// TwinCAT 3 PLC project Baustromverteiler
// ProgramVersion: 3.1.4023.0
// libraries:
//   EfficientIO Communicator, * (EfficientIO)
//   Lynus Energy Basic, * (Lynus AG)
//   Lynus Standards, * (Lynus AG)
//   Tc2_BABasic, * (Beckhoff Automation GmbH)
//   Tc2_Standard, * (Beckhoff Automation GmbH)
//   Tc2_System, * (Beckhoff Automation GmbH)
//   Tc2_Utilities, * (Beckhoff Automation GmbH)
//   Tc3_IotBase, * (Beckhoff Automation GmbH)
//   Tc3_JsonXml, * (Beckhoff Automation GmbH)
//   Tc3_Module, * (Beckhoff Automation GmbH)
// project tree:
//   / FastTask.TcTTO (not stored), GlobalTextList.TcGTLO, MiddleTask.TcTTO, SlowTask.TcTTO (not stored)
//   FBs/ FB_Enphase.TcPOU, FB_Enphase_Helper.TcPOU, FB_Shelly_Pro4PM.TcPOU, FB_Shelly_Pro4PM_Helper.TcPOU
//   POUs/ prgContactors.TcPOU, prgEM.TcPOU, prgEnphase.TcPOU, prgGrid.TcPOU, prgShelly1.TcPOU, prgShelly2.TcPOU, prgComEffIO.TcPOU, prgRWEffIO.TcPOU, prgSystemTime.TcPOU, prgVarEffIO.TcPOU (not stored)
// real-time tasks:
//   TASK FastTask: cycle T#5ms, priority 6, ADS port 350
//   TASK MiddleTask: cycle T#10ms, priority 8, ADS port 351
//   TASK SlowTask: cycle T#20ms, priority 10, ADS port 352
// I/O:
//   DEVICE Device 1 (Beckhoff CCAT)
//   DEVICE Device 2 (CX-BK)
//     Box 1 (CX-BK)
// variable links:
//   Baustromverteiler/Baustromverteiler Instance <-> Device 2 (CX-BK)/Box 1 (CX-BK)
//     MiddleTask Inputs/prgEM.fbEM1.fbKL3403.byStateCH1 <-> Term 3 (KL3403)/Channel 1/State
//     MiddleTask Inputs/prgEM.fbEM1.fbKL3403.byStateCH2 <-> Term 3 (KL3403)/Channel 2/State
//     MiddleTask Inputs/prgEM.fbEM1.fbKL3403.byStateCH3 <-> Term 3 (KL3403)/Channel 3/State
//     MiddleTask Inputs/prgEM.fbEM3.fbKL3403.byStateCH1 <-> Term 5 (KL3403)/Channel 1/State
//     MiddleTask Inputs/prgEM.fbEM3.fbKL3403.byStateCH2 <-> Term 5 (KL3403)/Channel 2/State
//     MiddleTask Inputs/prgEM.fbEM3.fbKL3403.byStateCH3 <-> Term 5 (KL3403)/Channel 3/State
//     MiddleTask Inputs/prgEM.fbEM1.fbKL3403.iDataInCH1 <-> Term 3 (KL3403)/Channel 1/Data In
//     MiddleTask Inputs/prgEM.fbEM1.fbKL3403.iDataInCH2 <-> Term 3 (KL3403)/Channel 2/Data In
//     MiddleTask Inputs/prgEM.fbEM1.fbKL3403.iDataInCH3 <-> Term 3 (KL3403)/Channel 3/Data In
//     MiddleTask Inputs/prgEM.fbEM3.fbKL3403.iDataInCH1 <-> Term 5 (KL3403)/Channel 1/Data In
//     MiddleTask Inputs/prgEM.fbEM3.fbKL3403.iDataInCH2 <-> Term 5 (KL3403)/Channel 2/Data In
//     MiddleTask Inputs/prgEM.fbEM3.fbKL3403.iDataInCH3 <-> Term 5 (KL3403)/Channel 3/Data In
//     MiddleTask Inputs/prgEM.fbKBusState.uiKBusState_OUT <-> Inputs/State
//     MiddleTask Outputs/prgContactors.bCircle6Switch <-> Term 2 (KL2408)/Channel 1/Output
//     MiddleTask Outputs/prgContactors.bCircle7Switch <-> Term 2 (KL2408)/Channel 3/Output
//     MiddleTask Outputs/prgEM.fbEM1.fbKL3403.byCntrCH1 <-> Term 3 (KL3403)/Channel 1/Ctrl
//     MiddleTask Outputs/prgEM.fbEM1.fbKL3403.byCntrCH2 <-> Term 3 (KL3403)/Channel 2/Ctrl
//     MiddleTask Outputs/prgEM.fbEM1.fbKL3403.byCntrCH3 <-> Term 3 (KL3403)/Channel 3/Ctrl
//     MiddleTask Outputs/prgEM.fbEM3.fbKL3403.byCntrCH1 <-> Term 5 (KL3403)/Channel 1/Ctrl
//     MiddleTask Outputs/prgEM.fbEM3.fbKL3403.byCntrCH2 <-> Term 5 (KL3403)/Channel 2/Ctrl
//     MiddleTask Outputs/prgEM.fbEM3.fbKL3403.byCntrCH3 <-> Term 5 (KL3403)/Channel 3/Ctrl

CONFIGURATION Baustromverteiler
    RESOURCE PLC ON TwinCAT3
        TASK MiddleTask(INTERVAL := T#10ms, PRIORITY := 8);
        PROGRAM prgContactors WITH MiddleTask : prgContactors;
        PROGRAM prgEM WITH MiddleTask : prgEM;
        PROGRAM prgShelly1 WITH MiddleTask : prgShelly1;
        PROGRAM prgShelly2 WITH MiddleTask : prgShelly2;
        PROGRAM prgSystemTime WITH MiddleTask : prgSystemTime;
        PROGRAM prgEnphase WITH MiddleTask : prgEnphase;
        PROGRAM prgGrid WITH MiddleTask : prgGrid;
    END_RESOURCE
END_CONFIGURATION

// ---- POUs/prgContactors.TcPOU
PROGRAM prgContactors
VAR
	bCircle6On				: BOOL;						//{#lynus.ag#()}
	bCircle6Off				: BOOL;						//{#lynus.ag#()}
	bCircle7On				: BOOL;						//{#lynus.ag#()}
	bCircle7Off				: BOOL;						//{#lynus.ag#()}
	bCircle6Switch	AT%Q*	: BOOL;						//{#lynus.ag#()}
	bCircle7Switch	AT%Q*	: BOOL;						//{#lynus.ag#()}
	fbCircle6				: FB_Light;
	fbCircle7				: FB_Light;
END_VAR

fbCircle6(bOn:=bCircle6On, bOff:=bCircle6Off, bLight=>bCircle6Switch);

fbCircle7(bOn:=bCircle7On, bOff:=bCircle7Off, bLight=>bCircle7Switch);

END_PROGRAM

// ---- POUs/prgEM.TcPOU
PROGRAM prgEM
VAR
	fbKBusState		: FB_K_Bus_State;
	fbEM1			: FB_EM_Beckhoff_KL3403;
	fbEM1Counter	: FB_EnergyCounter;
	fbEM2			: FB_EM_Beckhoff_KL3403;
	fbEM2Counter	: FB_EnergyCounter;
	fbEM3			: FB_EM_Beckhoff_KL3403;
	fbEM3Counter	: FB_EnergyCounter;
	fbC5Counter		: FB_EnergyCounter;
	lrPowerEM1		: LREAL;						//{#lynus.ag#()}
	lrPowerEM2		: LREAL;						//{#lynus.ag#()}
	lrPowerEM3		: LREAL;						//{#lynus.ag#()}
	lrPowerC5		: LREAL;						//{#lynus.ag#()}
END_VAR
VAR PERSISTENT
	lrCounterEM1	: LREAL;						//{#lynus.ag#()}
	lrCounterEM2	: LREAL;						//{#lynus.ag#()}
	lrCounterEM3	: LREAL;						//{#lynus.ag#()}
	lrCounterC5		: LREAL;						//{#lynus.ag#()}
END_VAR

fbKBusState(uiKBusState_OUT=> );

// Base Connection

fbEM1(
	bEnable:= TRUE, 
	bChannel1Invers:= TRUE,
	bChannel2Invers:= TRUE,
	bChannel3Invers:= TRUE,
	uiCurrentTransformerRatioL1:= 64, 
	uiCurrentTransformerRatioL2:= 64, 
	uiCurrentTransformerRatioL3:= 64, 
	uiKBusState_IN:= fbKBusState.uiKBusState_OUT, 
	stDataEMPower=> , 
	stDataEMCounter=> , 
	stDataEMPowerRealTime=> , 
	stDataEMCounterRealTime=> , 
	diNrOfEM_OUT=> );

lrPowerEM1 := fbEM1.stDataEMPower.lrPowerTotal;	

fbEM1Counter(
	byActiveTariff:= 1, 
	lrPowerInput:= lrPowerEM1, 
	lrTotalCounterEnergy_Consumption=> , 
	lrTotalCounterEnergy_Production=> , 
	lrCounterEnergyT1_Consumption=> , 
	lrCounterEnergyT2_Consumption=> , 
	lrCounterEnergyT1_Production=> , 
	lrCounterEnergyT2_Production=> );
	
IF fbEM1Counter.lrTotalCounterEnergy_Consumption > lrCounterEM1 THEN  	
	lrCounterEM1 := fbEM1Counter.lrTotalCounterEnergy_Consumption;
END_IF


// Circle6, 400V/32A

fbEM2(
	bEnable:= TRUE, 
	bChannel1Invers:= TRUE,
	bChannel2Invers:= TRUE,
	bChannel3Invers:= TRUE,
	uiCurrentTransformerRatioL1:= 35, 
	uiCurrentTransformerRatioL2:= 35, 
	uiCurrentTransformerRatioL3:= 35, 
	uiKBusState_IN:= fbKBusState.uiKBusState_OUT, 
	stDataEMPower=> , 
	stDataEMCounter=> , 
	stDataEMPowerRealTime=> , 
	stDataEMCounterRealTime=> , 
	diNrOfEM_OUT=> );

lrPowerEM2 := fbEM2.stDataEMPower.lrPowerTotal;	

fbEM2Counter(
	byActiveTariff:= 1, 
	lrPowerInput:= lrPowerEM2, 
	lrTotalCounterEnergy_Consumption=> , 
	lrTotalCounterEnergy_Production=> , 
	lrCounterEnergyT1_Consumption=> , 
	lrCounterEnergyT2_Consumption=> , 
	lrCounterEnergyT1_Production=> , 
	lrCounterEnergyT2_Production=> );
	
IF fbEM2Counter.lrTotalCounterEnergy_Consumption > lrCounterEM2 THEN  	
	lrCounterEM2 := fbEM2Counter.lrTotalCounterEnergy_Consumption;
END_IF


// Circle7, 400V/32A

fbEM3(
	bEnable:= TRUE, 
	bChannel1Invers:= FALSE,
	bChannel2Invers:= FALSE,
	bChannel3Invers:= FALSE,
	uiCurrentTransformerRatioL1:= 100, 
	uiCurrentTransformerRatioL2:= 100, 
	uiCurrentTransformerRatioL3:= 100, 
	uiKBusState_IN:= fbKBusState.uiKBusState_OUT, 
	stDataEMPower=> , 
	stDataEMCounter=> , 
	stDataEMPowerRealTime=> , 
	stDataEMCounterRealTime=> , 
	diNrOfEM_OUT=> );

lrPowerEM3 := fbEM3.stDataEMPower.lrPowerTotal;	

fbEM3Counter(
	byActiveTariff:= 1, 
	lrPowerInput:= lrPowerEM3, 
	lrTotalCounterEnergy_Consumption=> , 
	lrTotalCounterEnergy_Production=> , 
	lrCounterEnergyT1_Consumption=> , 
	lrCounterEnergyT2_Consumption=> , 
	lrCounterEnergyT1_Production=> , 
	lrCounterEnergyT2_Production=> );
	
IF fbEM3Counter.lrTotalCounterEnergy_Consumption > lrCounterEM3 THEN  	
	lrCounterEM3 := fbEM3Counter.lrTotalCounterEnergy_Consumption;
END_IF


// Circle5, 400V/16A

IF lrPowerEM1 - (lrPowerEM2 + lrPowerEM3 + prgShelly1.lrPowerC1 + prgShelly1.lrPowerC2 + prgShelly2.lrPowerC3 + prgShelly2.lrPowerC4) >= 0 THEN  	
	lrPowerC5 := lrPowerEM1 - (lrPowerEM2 + lrPowerEM3 + prgShelly1.lrPowerC1 + prgShelly1.lrPowerC2 + prgShelly2.lrPowerC3 + prgShelly2.lrPowerC4);
	ELSE
		lrPowerC5 := 0;
END_IF

fbC5Counter(
	byActiveTariff:= 1, 
	lrPowerInput:= lrPowerC5, 
	lrTotalCounterEnergy_Consumption=> , 
	lrTotalCounterEnergy_Production=> , 
	lrCounterEnergyT1_Consumption=> , 
	lrCounterEnergyT2_Consumption=> , 
	lrCounterEnergyT1_Production=> , 
	lrCounterEnergyT2_Production=> );
	
IF fbC5Counter.lrTotalCounterEnergy_Consumption > lrCounterC5 THEN  	
	lrCounterC5 := fbC5Counter.lrTotalCounterEnergy_Consumption;
END_IF

END_PROGRAM

// ---- POUs/prgShelly1.TcPOU
PROGRAM prgShelly1
VAR
	fbShelly1					: FB_Shelly_Pro4PM;
	// Circle1, 230V
	lrPowerC1					: LREAL;	//{#lynus.ag#()}
	lrVoltageC1					: LREAL;	//{#lynus.ag#()}
	lrEnergyC1					: LREAL;	//{#lynus.ag#()}
	lrPowerC1_W					: LREAL;
	lrEnergyC1_Wh				: LREAL;
	bCircle1On					: BOOL;		//{#lynus.ag#()}
	bCircle1Off					: BOOL;		//{#lynus.ag#()}
	bCircle1Switch				: BOOL;		//{#lynus.ag#()}

	// Circle2, 230V
	lrPowerC2					: LREAL;	//{#lynus.ag#()}
	lrVoltageC2					: LREAL;	//{#lynus.ag#()}
	lrEnergyC2					: LREAL;	//{#lynus.ag#()}
	lrPowerC2_W					: LREAL;
	lrEnergyC2_Wh				: LREAL;
	bCircle2On					: BOOL;		//{#lynus.ag#()}
	bCircle2Off					: BOOL;		//{#lynus.ag#()}
	bCircle2Switch				: BOOL;		//{#lynus.ag#()}
END_VAR

VAR PERSISTENT
// trigger command execution
	bEnableShelly1				: BOOL;		//{#lynus.ag#()}
END_VAR

fbShelly1(
	bStart:= bEnableShelly1, 
	tDelayRequest:= T#3S, 
	sHostname:= '192.168.1.20', 
	bValidResult=> , 
	bBusy=> , 
	bError=> , 
	bDone=> , 
	hrErrorCode=> ,
	lrpowerP1=> lrPowerC1_W, 
	lrvoltageP1=> lrVoltageC1, 
	lrenergyP1=> lrEnergyC1_Wh,
	lrpowerP2=> lrPowerC2_W, 
	lrvoltageP2=> lrVoltageC2, 
	lrenergyP2=> lrEnergyC2_Wh,
	bOnP1:= bCircle1On,
	bOffP1:= bCircle1Off,
	bStateP1=> bCircle1Switch,
	bOnP2:= bCircle2On,
	bOffP2:= bCircle2Off,
	bStateP2=> bCircle2Switch );

// re-calc Power to kW / kWh
lrPowerC1 := lrPowerC1_W / 1000;
lrPowerC2 := lrPowerC2_W / 1000;
lrEnergyC1 := lrEnergyC1_Wh / 1000;
lrEnergyC2 := lrEnergyC2_Wh / 1000;

END_PROGRAM

// ---- FBs/FB_Shelly_Pro4PM.TcPOU
FUNCTION_BLOCK FB_Shelly_Pro4PM
VAR_INPUT
	bStart				: BOOL;
	tDelayRequest		: TIME := T#3S;		//Timer for delay before start with the next read or write Request
	sHostname			: STRING(255);		//Hostname or IP Adress from the Server
	bOnP1				: BOOL;
	bOffP1				: BOOL;
	bOnP2				: BOOL;
	bOffP2				: BOOL;
	bOnP3				: BOOL;
	bOffP3				: BOOL;
	bOnP4				: BOOL;
	bOffP4				: BOOL;
END_VAR

VAR_IN_OUT
END_VAR

VAR_OUTPUT
	bValidResult				: BOOL;															//Valid Result received from Server
    bBusy						: BOOL;															//Function is Busy
    bError						: BOOL;															//Error sucess
	bDone						: BOOL;															//True after the decoding from the received Json File
	bConnected					: BOOL;															//Connection to the Server
	lrpowerP1					: LREAL;														//Received Value
	lrvoltageP1					: LREAL;														//Received Value
	lrenergyP1					: LREAL;														//Received Value
	lrpowerP2					: LREAL;														//Received Value
	lrvoltageP2					: LREAL;														//Received Value
	lrenergyP2					: LREAL;
	lrpowerP3					: LREAL;														//Received Value
	lrvoltageP3					: LREAL;														//Received Value
	lrenergyP3					: LREAL;
	lrpowerP4					: LREAL;														//Received Value
	lrvoltageP4					: LREAL;														//Received Value
	lrenergyP4					: LREAL;	
	hrErrorCode       			: HRESULT;														//Error Result from Http Client
	bStateP1					: BOOL;
	bStateP2					: BOOL;
	bStateP3					: BOOL;
	bStateP4					: BOOL;
END_VAR

VAR
	fbClient					: FB_IotHttpClient;
	fbHttpGet					: FB_Shelly_Pro4PM_Helper;
	timStartRequest				: TON;															//Timer to Start the Request
	FPStartRequest				: R_TRIG;														//Internal positive Edge
	FPDone						: R_TRIG;														//Internal positive Edge
	FNStart						: F_TRIG;														//Internal negative Edge
	SwitchOnP1					: R_TRIG;
	SwitchOffP1					: R_TRIG;
	SwitchOnP2					: R_TRIG;
	SwitchOffP2					: R_TRIG;
	SwitchOnP3					: R_TRIG;
	SwitchOffP3					: R_TRIG;
	SwitchOnP4					: R_TRIG;
	SwitchOffP4					: R_TRIG;
END_VAR

(*------------------------------------------------------------------------------------Configure HTTP Client------------------------------------------------------------------------------------------------------*)

fbClient.sHostName := sHostname;
fbClient.tConnectionTimeout := tDelayRequest;

IF NOT fbClient.bConfigured THEN 
	fbClient.nHostPort:= 80;
	fbClient.bKeepAlive := TRUE;
	fbClient.tConnectionTimeout := T#2S;
END_IF


//Timer to start the Request
FPStartRequest(CLK:= bStart, Q=> );
	timStartRequest(IN:= fbClient.bConfigured AND bStart AND NOT timStartRequest.Q, PT:= tDelayRequest, Q=> , ET=> );
		IF ((timStartRequest.Q AND NOT bBusy) OR (FPStartRequest.Q AND NOT bBusy AND fbClient.bConfigured)) THEN fbHttpGet.bSend := TRUE; END_IF

				
//Http Get Function
fbHttpGet(
	lrapowerP1 => lrpowerP1, 
	lrvoltageP1 => lrvoltageP1, 
	lraenergyP1 => lrenergyP1,
	lrapowerP2 => lrpowerP2, 
	lrvoltageP2 => lrvoltageP2, 
	lraenergyP2 => lrenergyP2,
	lrapowerP3 => lrpowerP3, 
	lrvoltageP3 => lrvoltageP3, 
	lraenergyP3 => lrenergyP3,
	lrapowerP4 => lrpowerP4, 
	lrvoltageP4 => lrvoltageP4, 
	lraenergyP4 => lrenergyP4, 
	bSend:= , 
	fbClient:= fbClient, 
	bBusy=> bBusy, 
	bError=> ,
	sContentS0=> ,
	sContentS1=> ,
	sContentS2=> ,
	sContentS3=> ,
	bStateP1=>bStateP1,
	bStateP2=>bStateP2,
	bStateP3=>bStateP3,
	bStateP4=>bStateP4 );


fbHttpGet.bSend := FALSE;

FPDone(CLK:= bDone, Q=> );

(*
//Http Client
FNStart(CLK:= bStart, Q=> );
	IF FNStart.Q THEN fbClient.Disconnect(); END_IF
*)

fbClient.Execute();

//Error
IF fbHttpGet.bError OR fbClient.bError THEN bError := TRUE; ELSE bError := FALSE; END_IF	
	hrErrorCode := fbClient.hrErrorCode;
	

// Relay Control, Switch P1
SwitchOnP1(CLK:=bOnP1);
IF SwitchOnP1.Q THEN
	fbHttpGet.bSetOnP1 := TRUE;
END_IF

SwitchOffP1(CLK:=bOffP1);
IF SwitchOffP1.Q THEN
	fbHttpGet.bSetOffP1 := TRUE;
END_IF

// Relay Control, Switch P2
SwitchOnP2(CLK:=bOnP2);
IF SwitchOnP2.Q THEN
	fbHttpGet.bSetOnP2 := TRUE;
END_IF

SwitchOffP2(CLK:=bOffP2);
IF SwitchOffP2.Q THEN
	fbHttpGet.bSetOffP2 := TRUE;
END_IF

// Relay Control, Switch P3
SwitchOnP3(CLK:=bOnP3);
IF SwitchOnP3.Q THEN
	fbHttpGet.bSetOnP3 := TRUE;
END_IF

SwitchOffP3(CLK:=bOffP3);
IF SwitchOffP3.Q THEN
	fbHttpGet.bSetOffP3 := TRUE;
END_IF

// Relay Control, Switch P4
SwitchOnP4(CLK:=bOnP4);
IF SwitchOnP4.Q THEN
	fbHttpGet.bSetOnP4 := TRUE;
END_IF

SwitchOffP4(CLK:=bOffP4);
IF SwitchOffP4.Q THEN
	fbHttpGet.bSetOffP4 := TRUE;
END_IF

END_FUNCTION_BLOCK

// ---- FBs/FB_Shelly_Pro4PM_Helper.TcPOU
FUNCTION_BLOCK FB_Shelly_Pro4PM_Helper
VAR_INPUT
	bSend			: BOOL;
	bSetOnP1		: BOOL;
	bSetOffP1		: BOOL;
	bSetOnP2		: BOOL;
	bSetOffP2		: BOOL;
	bSetOnP3		: BOOL;
	bSetOffP3		: BOOL;
	bSetOnP4		: BOOL;
	bSetOffP4		: BOOL;
END_VAR

VAR_IN_OUT
	fbClient		: FB_IotHttpClient;
END_VAR

VAR_OUTPUT
	bBusy			: BOOL;
	bError			: BOOL;
	bStateP1		: BOOL;
	bStateP2		: BOOL;
	bStateP3		: BOOL;
	bStateP4		: BOOL;
	lrapowerP1		: LREAL;
	lrvoltageP1		: LREAL;
	lraenergyP1		: LREAL;
	lrapowerP2		: LREAL;
	lrvoltageP2		: LREAL;
	lraenergyP2		: LREAL;
	lrapowerP3		: LREAL;
	lrvoltageP3		: LREAL;
	lraenergyP3		: LREAL;
	lrapowerP4		: LREAL;
	lrvoltageP4		: LREAL;
	lraenergyP4		: LREAL;
END_VAR

VAR
	fbRequestSwitch0	: FB_IotHttpRequest;
	fbRequestSwitch1	: FB_IotHttpRequest;
	fbRequestSwitch2	: FB_IotHttpRequest;
	fbRequestSwitch3	: FB_IotHttpRequest;
	fbJson				: FB_JsonDomParser;
	nState				: UDINT;
	RisingEdge			: R_TRIG;
	RisingEdgeSetOnP1	: R_TRIG;
	RisingEdgeSetOffP1	: R_TRIG;
	RisingEdgeSetOnP2	: R_TRIG;
	RisingEdgeSetOffP2	: R_TRIG;
	RisingEdgeSetOnP3	: R_TRIG;
	RisingEdgeSetOffP3	: R_TRIG;
	RisingEdgeSetOnP4	: R_TRIG;
	RisingEdgeSetOffP4	: R_TRIG;
	timTimeout			: TON;
	tTimeOut			: TIME := T#30S;
	timTimeoutSwitch	: TON;
	tTimeOutSwitch		: TIME := T#5S;
	
	bGetContentResult	: BOOL;
	sContentS0			: STRING(511);
	sContentS1			: STRING(511);
	sContentS2			: STRING(511);
	sContentS3			: STRING(511);
	
	bGetJsonResult		: BOOL;
	jsonDoc				: SJsonValue;
	jsonVal				: SJsonValue;
	
	nReqCount			: UDINT;	
	nResCount			: UDINT;
	nValidResCount		: UDINT;
	nErrCount			: UDINT;
END_VAR

//Timer for Timeout
timTimeout(IN:= nState = 1 AND bBusy, PT:= tTimeOut, Q=> , ET=> );
	IF timTimeout.Q THEN 
		nState := 0;
		bBusy := FALSE;
	END_IF
	
timTimeoutSwitch(IN:= bSetOnP1 OR bSetOffP1 OR bSetOnP2 OR bSetOffP2 OR bSetOnP3 OR bSetOffP3 OR bSetOnP4 OR bSetOffP4, PT:= tTimeOut, Q=> , ET=> );
	IF timTimeoutSwitch.Q THEN 
		bSetOnP1 := FALSE;
		bSetOffP1 := FALSE;
		bSetOnP2 := FALSE;
		bSetOffP2 := FALSE;
		bSetOnP3 := FALSE;
		bSetOffP3 := FALSE;
		bSetOnP4 := FALSE;
		bSetOffP4 := FALSE;
	END_IF

RisingEdge(CLK:= bSend );
RisingEdgeSetOnP1(CLK:= bSetOnP1 );
RisingEdgeSetOffP1(CLK:= bSetOffP1 );
RisingEdgeSetOnP2(CLK:= bSetOnP2 );
RisingEdgeSetOffP2(CLK:= bSetOffP2 );
RisingEdgeSetOnP3(CLK:= bSetOnP3 );
RisingEdgeSetOffP3(CLK:= bSetOffP3 );
RisingEdgeSetOnP4(CLK:= bSetOnP4 );
RisingEdgeSetOffP4(CLK:= bSetOffP4 );

CASE nState OF
0:	
	IF RisingEdge.Q THEN 
		IF
			fbRequestSwitch0.SendRequest(sUri:='/rpc/Switch.GetStatus?id=0', fbClient:=fbClient, eRequestType:=ETcIotHttpRequestType.HTTP_Get, 0, 0, 0) AND
			fbRequestSwitch1.SendRequest(sUri:='/rpc/Switch.GetStatus?id=1', fbClient:=fbClient, eRequestType:=ETcIotHttpRequestType.HTTP_Get, 0, 0, 0) AND
			fbRequestSwitch2.SendRequest(sUri:='/rpc/Switch.GetStatus?id=2', fbClient:=fbClient, eRequestType:=ETcIotHttpRequestType.HTTP_Get, 0, 0, 0) AND
			fbRequestSwitch3.SendRequest(sUri:='/rpc/Switch.GetStatus?id=3', fbClient:=fbClient, eRequestType:=ETcIotHttpRequestType.HTTP_Get, 0, 0, 0) THEN				
			nState:= 1;
			nReqCount:= nReqCount+1;
			bBusy:= TRUE;
			bError:= FALSE;
		END_IF					
	END_IF
	
	IF RisingEdgeSetOnP1.Q THEN 
		IF
			fbRequestSwitch0.SendRequest(sUri:='/rpc/Switch.Set?id=0&on=true', fbClient:=fbClient, eRequestType:=ETcIotHttpRequestType.HTTP_Get, 0, 0, 0) THEN				
			bSetOnP1 := FALSE;
			nState:= 1;
			bBusy:= TRUE;
			bError:= FALSE;
		END_IF					
	END_IF
	
	IF RisingEdgeSetOffP1.Q THEN 
		IF
			fbRequestSwitch0.SendRequest(sUri:='/rpc/Switch.Set?id=0&on=false', fbClient:=fbClient, eRequestType:=ETcIotHttpRequestType.HTTP_Get, 0, 0, 0) THEN				
			bSetOffP1 := FALSE;
			nState:= 1;
			bBusy:= TRUE;
			bError:= FALSE;
		END_IF					
	END_IF
	
	IF RisingEdgeSetOnP2.Q THEN 
		IF
			fbRequestSwitch1.SendRequest(sUri:='/rpc/Switch.Set?id=1&on=true', fbClient:=fbClient, eRequestType:=ETcIotHttpRequestType.HTTP_Get, 0, 0, 0) THEN				
			bSetOnP2 := FALSE;
			nState:= 1;
			bBusy:= TRUE;
			bError:= FALSE;
		END_IF					
	END_IF
	
	IF RisingEdgeSetOffP2.Q THEN 
		IF
			fbRequestSwitch1.SendRequest(sUri:='/rpc/Switch.Set?id=1&on=false', fbClient:=fbClient, eRequestType:=ETcIotHttpRequestType.HTTP_Get, 0, 0, 0) THEN				
			bSetOffP2 := FALSE;
			nState:= 1;
			bBusy:= TRUE;
			bError:= FALSE;
		END_IF					
	END_IF
	
	IF RisingEdgeSetOnP3.Q THEN 
		IF
			fbRequestSwitch2.SendRequest(sUri:='/rpc/Switch.Set?id=2&on=true', fbClient:=fbClient, eRequestType:=ETcIotHttpRequestType.HTTP_Get, 0, 0, 0) THEN				
			bSetOnP3 := FALSE;
			nState:= 1;
			bBusy:= TRUE;
			bError:= FALSE;
		END_IF					
	END_IF
	
	IF RisingEdgeSetOffP3.Q THEN 
		IF
			fbRequestSwitch2.SendRequest(sUri:='/rpc/Switch.Set?id=2&on=false', fbClient:=fbClient, eRequestType:=ETcIotHttpRequestType.HTTP_Get, 0, 0, 0) THEN				
			bSetOffP3 := FALSE;
			nState:= 1;
			bBusy:= TRUE;
			bError:= FALSE;
		END_IF					
	END_IF
	
	IF RisingEdgeSetOnP4.Q THEN 
		IF
			fbRequestSwitch3.SendRequest(sUri:='/rpc/Switch.Set?id=3&on=true', fbClient:=fbClient, eRequestType:=ETcIotHttpRequestType.HTTP_Get, 0, 0, 0) THEN				
			bSetOnP4 := FALSE;
			nState:= 1;
			bBusy:= TRUE;
			bError:= FALSE;
		END_IF					
	END_IF
	
	IF RisingEdgeSetOffP4.Q THEN 
		IF
			fbRequestSwitch3.SendRequest(sUri:='/rpc/Switch.Set?id=3&on=false', fbClient:=fbClient, eRequestType:=ETcIotHttpRequestType.HTTP_Get, 0, 0, 0) THEN				
			bSetOffP4 := FALSE;
			nState:= 1;
			bBusy:= TRUE;
			bError:= FALSE;
		END_IF					
	END_IF
	
1:
	IF NOT fbRequestSwitch0.bBusy AND NOT fbRequestSwitch1.bBusy AND NOT fbRequestSwitch2.bBusy AND NOT fbRequestSwitch3.bBusy THEN
		bError:= TRUE;
		
		IF NOT fbRequestSwitch0.bError THEN				 
			bGetContentResult:= fbRequestSwitch0.GetContent(pContent:= ADR(sContentS0), nContentSize:= SIZEOF(sContentS0), bSetNullTermination:= TRUE);
			IF fbRequestSwitch0.nStatusCode >= 200 AND fbRequestSwitch0.nStatusCode < 300 THEN
				bGetJsonResult:= FALSE;
				jsonDoc:= fbRequestSwitch0.GetJsonDomContent(fbJson);
				IF jsonDoc <> 0 THEN
					bGetJsonResult:= TRUE;
					IF fbJson.HasMember(jsonDoc, 'output')  THEN
						jsonVal:= fbJson.FindMember(jsonDoc, 'output');
						nValidResCount:= nValidResCount+1;					
						IF fbJson.IsBool(jsonVal) THEN							
							bStateP1:= fbJson.GetBool(jsonVal);									
						END_IF
						jsonVal:= fbJson.FindMember(jsonDoc, 'apower');
						nValidResCount:= nValidResCount+1;
						IF fbJson.IsDouble(jsonVal) THEN							
							lrapowerP1:= fbJson.GetDouble(jsonVal);									
						END_IF
						jsonVal:= fbJson.FindMember(jsonDoc, 'voltage');
						nValidResCount:= nValidResCount+1;					
						IF fbJson.IsDouble(jsonVal) THEN							
							lrvoltageP1:= fbJson.GetDouble(jsonVal);									
						END_IF
						jsonVal:= fbJson.FindMember(jsonDoc, 'aenergy');
                        IF fbJson.HasMember(jsonVal, 'total') THEN
                            jsonVal:= fbJson.FindMember(jsonVal, 'total');
                            nValidResCount:= nValidResCount+1;
                            IF fbJson.IsDouble(jsonVal) THEN
                                lraenergyP1:= fbJson.GetDouble(jsonVal);
                            END_IF
						bError:= FALSE;
						END_IF
					END_IF						
				nResCount:= nResCount+1;			
				END_IF
			END_IF
		END_IF
		
		IF NOT fbRequestSwitch1.bError THEN				 
			bGetContentResult:= fbRequestSwitch1.GetContent(pContent:= ADR(sContentS1), nContentSize:= SIZEOF(sContentS1), bSetNullTermination:= TRUE);
			IF fbRequestSwitch1.nStatusCode >= 200 AND fbRequestSwitch1.nStatusCode < 300 THEN
				bGetJsonResult:= FALSE;
				jsonDoc:= fbRequestSwitch1.GetJsonDomContent(fbJson);
				IF jsonDoc <> 0 THEN
					bGetJsonResult:= TRUE;
					IF fbJson.HasMember(jsonDoc, 'output')  THEN
						jsonVal:= fbJson.FindMember(jsonDoc, 'output');
						nValidResCount:= nValidResCount+1;					
						IF fbJson.IsBool(jsonVal) THEN							
							bStateP2:= fbJson.GetBool(jsonVal);									
						END_IF
						jsonVal:= fbJson.FindMember(jsonDoc, 'apower');
						nValidResCount:= nValidResCount+1;
						IF fbJson.IsDouble(jsonVal) THEN							
							lrapowerP2:= fbJson.GetDouble(jsonVal);									
						END_IF
						jsonVal:= fbJson.FindMember(jsonDoc, 'voltage');
						nValidResCount:= nValidResCount+1;					
						IF fbJson.IsDouble(jsonVal) THEN							
							lrvoltageP2:= fbJson.GetDouble(jsonVal);									
						END_IF
						jsonVal:= fbJson.FindMember(jsonDoc, 'aenergy');
                        IF fbJson.HasMember(jsonVal, 'total') THEN
                            jsonVal:= fbJson.FindMember(jsonVal, 'total');
                            nValidResCount:= nValidResCount+1;
                            IF fbJson.IsDouble(jsonVal) THEN
                                lraenergyP2:= fbJson.GetDouble(jsonVal);
                            END_IF
						bError:= FALSE;
						END_IF
					END_IF						
				nResCount:= nResCount+1;			
				END_IF
			END_IF
		END_IF
		
		IF NOT fbRequestSwitch2.bError THEN				 
			bGetContentResult:= fbRequestSwitch2.GetContent(pContent:= ADR(sContentS2), nContentSize:= SIZEOF(sContentS2), bSetNullTermination:= TRUE);
			IF fbRequestSwitch2.nStatusCode >= 200 AND fbRequestSwitch2.nStatusCode < 300 THEN
				bGetJsonResult:= FALSE;
				jsonDoc:= fbRequestSwitch2.GetJsonDomContent(fbJson);
				IF jsonDoc <> 0 THEN
					bGetJsonResult:= TRUE;
					IF fbJson.HasMember(jsonDoc, 'output')  THEN
						jsonVal:= fbJson.FindMember(jsonDoc, 'output');
						nValidResCount:= nValidResCount+1;					
						IF fbJson.IsBool(jsonVal) THEN							
							bStateP3:= fbJson.GetBool(jsonVal);									
						END_IF
						jsonVal:= fbJson.FindMember(jsonDoc, 'apower');
						nValidResCount:= nValidResCount+1;
						IF fbJson.IsDouble(jsonVal) THEN							
							lrapowerP3:= fbJson.GetDouble(jsonVal);									
						END_IF
						jsonVal:= fbJson.FindMember(jsonDoc, 'voltage');
						nValidResCount:= nValidResCount+1;					
						IF fbJson.IsDouble(jsonVal) THEN							
							lrvoltageP3:= fbJson.GetDouble(jsonVal);									
						END_IF
						jsonVal:= fbJson.FindMember(jsonDoc, 'aenergy');
                        IF fbJson.HasMember(jsonVal, 'total') THEN
                            jsonVal:= fbJson.FindMember(jsonVal, 'total');
                            nValidResCount:= nValidResCount+1;
                            IF fbJson.IsDouble(jsonVal) THEN
                                lraenergyP3:= fbJson.GetDouble(jsonVal);
                            END_IF
						bError:= FALSE;
						END_IF
					END_IF						
				nResCount:= nResCount+1;			
				END_IF
			END_IF
		END_IF
		
		IF NOT fbRequestSwitch3.bError THEN				 
			bGetContentResult:= fbRequestSwitch3.GetContent(pContent:= ADR(sContentS3), nContentSize:= SIZEOF(sContentS3), bSetNullTermination:= TRUE);
			IF fbRequestSwitch3.nStatusCode >= 200 AND fbRequestSwitch3.nStatusCode < 300 THEN
				bGetJsonResult:= FALSE;
				jsonDoc:= fbRequestSwitch3.GetJsonDomContent(fbJson);
				IF jsonDoc <> 0 THEN
					bGetJsonResult:= TRUE;
					IF fbJson.HasMember(jsonDoc, 'output')  THEN
						jsonVal:= fbJson.FindMember(jsonDoc, 'output');
						nValidResCount:= nValidResCount+1;					
						IF fbJson.IsBool(jsonVal) THEN							
							bStateP4:= fbJson.GetBool(jsonVal);									
						END_IF
						jsonVal:= fbJson.FindMember(jsonDoc, 'apower');
						nValidResCount:= nValidResCount+1;
						IF fbJson.IsDouble(jsonVal) THEN							
							lrapowerP4:= fbJson.GetDouble(jsonVal);									
						END_IF
						jsonVal:= fbJson.FindMember(jsonDoc, 'voltage');
						nValidResCount:= nValidResCount+1;					
						IF fbJson.IsDouble(jsonVal) THEN							
							lrvoltageP4:= fbJson.GetDouble(jsonVal);									
						END_IF
						jsonVal:= fbJson.FindMember(jsonDoc, 'aenergy');
                        IF fbJson.HasMember(jsonVal, 'total') THEN
                            jsonVal:= fbJson.FindMember(jsonVal, 'total');
                            nValidResCount:= nValidResCount+1;
                            IF fbJson.IsDouble(jsonVal) THEN
                                lraenergyP4:= fbJson.GetDouble(jsonVal);
                            END_IF
						bError:= FALSE;
						END_IF
					END_IF						
				nResCount:= nResCount+1;			
				END_IF
			END_IF
		END_IF
		
	nState:= 0;
	bBusy:= FALSE;
		IF bError THEN
			nErrCount:= nErrCount+1;
		END_IF
	END_IF
	
END_CASE

END_FUNCTION_BLOCK

// ---- POUs/prgShelly2.TcPOU
PROGRAM prgShelly2
VAR
	fbShelly2					: FB_Shelly_Pro4PM;
	// Circle3, 230V
	lrPowerC3					: LREAL;	//{#lynus.ag#()}
	lrVoltageC3					: LREAL;	//{#lynus.ag#()}
	lrEnergyC3					: LREAL;	//{#lynus.ag#()}
	lrPowerC3_W					: LREAL;
	lrEnergyC3_Wh				: LREAL;
	bCircle3On					: BOOL;		//{#lynus.ag#()}
	bCircle3Off					: BOOL;		//{#lynus.ag#()}
	bCircle3Switch				: BOOL;		//{#lynus.ag#()}

	// Circle4, 230V
	lrPowerC4					: LREAL;	//{#lynus.ag#()}
	lrVoltageC4					: LREAL;	//{#lynus.ag#()}
	lrEnergyC4					: LREAL;	//{#lynus.ag#()}
	lrPowerC4_W					: LREAL;
	lrEnergyC4_Wh				: LREAL;
	bCircle4On					: BOOL;		//{#lynus.ag#()}
	bCircle4Off					: BOOL;		//{#lynus.ag#()}
	bCircle4Switch				: BOOL;		//{#lynus.ag#()}
	
	fbTimerC4					: FB_WeeklyTimeSwitch;
	fbCalcSunriseSunset   		: FB_CalcSunriseSunset;
	todSunrise            		: TOD;
	todSunset             		: TOD;
END_VAR
VAR PERSISTENT
// trigger command execution
	bEnableShelly2				: BOOL;		//{#lynus.ag#()}
	bEnableTimerC4				: BOOL;		//{#lynus.ag#()}
END_VAR

fbShelly2(
	bStart:= bEnableShelly2, 
	tDelayRequest:= T#3S, 
	sHostname:= '192.168.1.21', 
	bValidResult=> , 
	bBusy=> , 
	bError=> , 
	bDone=> , 
	hrErrorCode=> ,
	lrpowerP3=> lrPowerC3_W, 
	lrvoltageP3=> lrVoltageC3, 
	lrenergyP3=> lrEnergyC3,
	lrpowerP4=> lrPowerC4_W, 
	lrvoltageP4=> lrVoltageC4, 
	lrenergyP4=> lrEnergyC4,
	bOnP3:= bCircle3On,
	bOffP3:= bCircle3Off,
	bStateP3=> bCircle3Switch,
	bOnP4:= bCircle4On,
	bOffP4:= bCircle4Off,
	bStateP4=> bCircle4Switch );

// re-calc Power to kW
lrPowerC3 := lrPowerC3_W / 1000;
lrPowerC4 := lrPowerC4_W / 1000;
lrEnergyC3 := lrEnergyC3_Wh / 1000;
lrEnergyC4 := lrEnergyC4_Wh / 1000;


IF prgSystemTime.bSystemTimeValid THEN

	fbCalcSunriseSunset(
		fDegreeOfLongitude := 11.5820,   (* Longitude of Munich, Lochhausen *)
        fDegreeOfLatitude := 48.1351,   (* Latitude of Munich, Lochhausen *)
    	fReferenceMeridian := 15.0,  (* Central European Time *)
        dCurrentDate := DT_TO_DATE(prgSystemTime.dtSystemTime),
        todSunrise => todSunrise,
        todSunset => todSunset);
END_IF



IF prgSystemTime.bSystemTimeValid THEN

	fbTimerC4(
		bEnable:=bEnableTimerC4, 
		tCurrentDateTime:=prgSystemTime.dtSystemTime, 
		tSwitchOnTime:=todSunrise, 
		tSwitchOffTime:=todSunset, 
		bSunday:=TRUE, 
		bMonday:=TRUE, 
		bTuesday:=TRUE, 
		bWednesday:=TRUE, 
		bThursday:=TRUE, 
		bFriday:=TRUE, 
		bSaturday:=TRUE,
		bEdgeOn=> bCircle4On,
		bEdgeOff=> bCircle4Off);
END_IF

END_PROGRAM

// ---- POUs/prgSystemTime.TcPOU
PROGRAM prgSystemTime
VAR
	fbGetTime			: NT_GetTime;
	dtSystemTime		: DT;
	stDateTime			: TIMESTRUCT;
	tonGetTime			: TON;
	nStep				: INT;
	bSystemTimeValid	: BOOL := FALSE;
END_VAR

CASE nStep OF
0:
	tonGetTime(IN:=TRUE, PT:=T#500MS);
	IF (tonGetTime.Q) THEN
		tonGetTime(IN := FALSE);
		nStep:=10;
	END_IF

10:
	fbGetTime(NETID:='', START:=TRUE, TMOUT:=T#2S);
	IF (NOT fbGetTime.BUSY) THEN
		stDateTime := fbGetTime.TIMESTR;
		dtSystemTime := SYSTEMtimE_TO_DT(fbGetTime.TIMESTR);
		fbGetTime(START := FALSE);
		bSystemTimeValid := TRUE;
		nStep := 0;
	END_IF	
END_CASE

END_PROGRAM

// ---- POUs/prgEnphase.TcPOU
PROGRAM prgEnphase
VAR
	fbEnphase					: FB_Enphase;
	fbPVCounter					: FB_EnergyCounter;
	fbGridCounter				: FB_EnergyCounter;
	lrPowerPV_W					: LREAL;
	lrPowerGrid_W				: LREAL;
	lrPowerPV					: LREAL;						//{#lynus.ag#()}
	lrPowerGrid					: LREAL;						//{#lynus.ag#()}
	lrCO2PV						: LREAL;						//{#lynus.ag#()}
	lrTreePV					: LREAL;						//{#lynus.ag#()}
END_VAR

VAR PERSISTENT
// trigger command execution
	bEnableEnphase				: BOOL;							//{#lynus.ag#()}
	lrCounterPV					: LREAL;						//{#lynus.ag#()}
	lrCounterGrid				: LREAL;						//{#lynus.ag#()}
END_VAR

fbEnphase(
	bStart:= bEnableEnphase, 
	tDelayRequest:= T#3S, 
	sHostname:= '192.168.1.30', 
	bValidResult=> , 
	bBusy=> , 
	bError=> , 
	bDone=> , 
	hrErrorCode=> ,
	lrpowerprod => lrPowerPV_W,
	lrpowercons => lrPowerGrid_W );
	
// re-calc Power to kW
lrPowerPV := lrPowerPV_W / 1000;
lrPowerGrid := lrPowerGrid_W / 1000;

fbPVCounter(
	byActiveTariff:= 1, 
	lrPowerInput:= lrPowerPV, 
	lrTotalCounterEnergy_Consumption=> , 
	lrTotalCounterEnergy_Production=> , 
	lrCounterEnergyT1_Consumption=> , 
	lrCounterEnergyT2_Consumption=> , 
	lrCounterEnergyT1_Production=> , 
	lrCounterEnergyT2_Production=> );
	
IF fbPVCounter.lrTotalCounterEnergy_Consumption > lrCounterPV THEN  	
	lrCounterPV := fbPVCounter.lrTotalCounterEnergy_Consumption;
END_IF

lrCO2PV := lrCounterPV * 0.428;
lrTreePV := lrCO2PV / 12.5;

fbGridCounter(
	byActiveTariff:= 1, 
	lrPowerInput:= lrPowerGrid, 
	lrTotalCounterEnergy_Consumption=> , 
	lrTotalCounterEnergy_Production=> , 
	lrCounterEnergyT1_Consumption=> , 
	lrCounterEnergyT2_Consumption=> , 
	lrCounterEnergyT1_Production=> , 
	lrCounterEnergyT2_Production=> );
	
IF fbGridCounter.lrTotalCounterEnergy_Consumption > lrCounterGrid THEN  	
	lrCounterGrid := fbGridCounter.lrTotalCounterEnergy_Consumption;
END_IF

END_PROGRAM

// ---- FBs/FB_Enphase.TcPOU
FUNCTION_BLOCK FB_Enphase
VAR_INPUT
	bStart				: BOOL;
	tDelayRequest		: TIME := T#3S;		//Timer for delay before start with the next read or write Request
	sHostname			: STRING(255);		//Hostname or IP Adress from the Server
END_VAR

VAR_IN_OUT
END_VAR

VAR_OUTPUT
	bValidResult				: BOOL;															//Valid Result received from Server
    bBusy						: BOOL;															//Function is Busy
    bError						: BOOL;															//Error sucess
	bDone						: BOOL;															//True after the decoding from the received Json File
	bConnected					: BOOL;															//Connection to the Server
	lrpowerprod					: LREAL;														//Received Value
	lrpowercons					: LREAL;														//Received Value
	hrErrorCode       			: HRESULT;														//Error Result from Http Client
END_VAR

VAR
	fbClient					: FB_IotHttpClient;
	fbHttpGet					: FB_Enphase_Helper;
	timStartRequest				: TON;															//Timer to Start the Request
	FPStartRequest				: R_TRIG;														//Internal positive Edge
	FPDone						: R_TRIG;														//Internal positive Edge
	FNStart						: F_TRIG;														//Internal negative Edge
END_VAR

(*------------------------------------------------------------------------------------Configure HTTP Client------------------------------------------------------------------------------------------------------*)

fbClient.sHostName := sHostname;
fbClient.tConnectionTimeout := tDelayRequest;

IF NOT fbClient.bConfigured THEN 
	fbClient.nHostPort:= 80;
	fbClient.bKeepAlive := TRUE;
	fbClient.tConnectionTimeout := T#2S;
END_IF


//Timer to start the Request
FPStartRequest(CLK:= bStart, Q=> );
	timStartRequest(IN:= fbClient.bConfigured AND bStart AND NOT timStartRequest.Q, PT:= tDelayRequest, Q=> , ET=> );
		IF ((timStartRequest.Q AND NOT bBusy) OR (FPStartRequest.Q AND NOT bBusy AND fbClient.bConfigured)) THEN fbHttpGet.bSend := TRUE; END_IF

				
//Http Get Function
fbHttpGet(
	lrpowerprod => lrpowerprod, 
	lrpowercons => lrpowercons,
	bSend:= , 
	fbClient:= fbClient, 
	bBusy=> bBusy, 
	bError=> ,
	sContent=> );


fbHttpGet.bSend := FALSE;

FPDone(CLK:= bDone, Q=> );

(*
//Http Client
FNStart(CLK:= bStart, Q=> );
	IF FNStart.Q THEN fbClient.Disconnect(); END_IF
*)

fbClient.Execute();

//Error
IF fbHttpGet.bError OR fbClient.bError THEN bError := TRUE; ELSE bError := FALSE; END_IF	
	hrErrorCode := fbClient.hrErrorCode;

END_FUNCTION_BLOCK

// ---- FBs/FB_Enphase_Helper.TcPOU
FUNCTION_BLOCK FB_Enphase_Helper
VAR_INPUT
	bSend			: BOOL;
END_VAR

VAR_IN_OUT
	fbClient		: FB_IotHttpClient;
END_VAR

VAR_OUTPUT
	bBusy			: BOOL;
	bError			: BOOL;
	lrpowerprod			: LREAL;
	lrpowercons			: LREAL;

END_VAR

VAR
	fbRequestEnphase	: FB_IotHttpRequest;
	fbJson				: FB_JsonDomParser;
	nState				: UDINT;
	RisingEdge			: R_TRIG;
	timTimeout			: TON;
	tTimeOut			: TIME := T#30S;
	
	bGetContentResult	: BOOL;
	sContent			: STRING(2048);
	
	bGetJsonResult		: BOOL;
	jsonDoc				: SJsonValue;
	jsonVal				: SJsonValue;
	
	nReqCount			: UDINT;	
	nResCount			: UDINT;
	nValidResCount		: UDINT;
	nErrCount			: UDINT;
END_VAR

//Timer for Timeout
timTimeout(IN:= nState = 1 AND bBusy, PT:= tTimeOut, Q=> , ET=> );
	IF timTimeout.Q THEN 
		nState := 0;
		bBusy := FALSE;
	END_IF


RisingEdge(CLK:= bSend );


CASE nState OF
0:	
	IF RisingEdge.Q THEN 
		IF
			fbRequestEnphase.SendRequest(sUri:='/production.json', fbClient:=fbClient, eRequestType:=ETcIotHttpRequestType.HTTP_Get, 0, 0, 0) THEN				
				nState:= 1;
				nReqCount:= nReqCount+1;
				bBusy:= TRUE;
				bError:= FALSE;
		END_IF					
	END_IF
	
	
1:
	IF NOT fbRequestEnphase.bBusy THEN
		bError:= TRUE;
		
		IF NOT fbRequestEnphase.bError THEN				 
			bGetContentResult:= fbRequestEnphase.GetContent(pContent:= ADR(sContent), nContentSize:= SIZEOF(sContent), bSetNullTermination:= TRUE);
			IF fbRequestEnphase.nStatusCode >= 200 AND fbRequestEnphase.nStatusCode < 300 THEN
				bGetJsonResult:= FALSE;
				jsonDoc:= fbRequestEnphase.GetJsonDomContent(fbJson);
				IF jsonDoc <> 0 THEN
					bGetJsonResult:= TRUE;
					IF fbJson.HasMember(jsonDoc, 'production')  THEN
						jsonVal:= fbJson.FindMember(jsonDoc, 'production');
						jsonVal:= fbJson.GetArrayValueByIdx(jsonVal, 1);
                        IF fbJson.HasMember(jsonVal, 'wNow') THEN
                            jsonVal:= fbJson.FindMember(jsonVal, 'wNow');
                            nValidResCount:= nValidResCount+1;
                            IF fbJson.IsDouble(jsonVal) THEN
                                lrpowerprod:= fbJson.GetDouble(jsonVal);
                            END_IF
						bError:= FALSE;
						END_IF
					END_IF
					IF fbJson.HasMember(jsonDoc, 'consumption')  THEN
						jsonVal:= fbJson.FindMember(jsonDoc, 'consumption');
						jsonVal:= fbJson.GetArrayValueByIdx(jsonVal, 1);
                        IF fbJson.HasMember(jsonVal, 'wNow') THEN
                            jsonVal:= fbJson.FindMember(jsonVal, 'wNow');
                            nValidResCount:= nValidResCount+1;
                            IF fbJson.IsDouble(jsonVal) THEN
                                lrpowercons:= fbJson.GetDouble(jsonVal);
                            END_IF
						bError:= FALSE;
						END_IF
					END_IF						
				nResCount:= nResCount+1;			
				END_IF
			END_IF
		END_IF
		
	nState:= 0;
	bBusy:= FALSE;
		IF bError THEN
			nErrCount:= nErrCount+1;
		END_IF
	END_IF
	
END_CASE

END_FUNCTION_BLOCK

// ---- POUs/prgGrid.TcPOU
PROGRAM prgGrid
VAR
	fbGridCounter				: FB_EnergyCounter;
	lrPowerGrid					: LREAL;						//{#lynus.ag#()}
END_VAR
VAR PERSISTENT
	lrCounterGridProd			: LREAL;						//{#lynus.ag#()}
	lrCounterGridCon			: LREAL;						//{#lynus.ag#()}
END_VAR


lrPowerGrid := prgEM.lrPowerEM3 - prgEnphase.lrPowerPV;

fbGridCounter(
	byActiveTariff:= 1, 
	lrPowerInput:= lrPowerGrid, 
	lrTotalCounterEnergy_Consumption=> , 
	lrTotalCounterEnergy_Production=> , 
	lrCounterEnergyT1_Consumption=> , 
	lrCounterEnergyT2_Consumption=> , 
	lrCounterEnergyT1_Production=> , 
	lrCounterEnergyT2_Production=> );
	
IF fbGridCounter.lrTotalCounterEnergy_Consumption > lrCounterGridCon THEN  	
	lrCounterGridCon := fbGridCounter.lrTotalCounterEnergy_Consumption;
END_IF
	IF fbGridCounter.lrTotalCounterEnergy_Production > lrCounterGridProd THEN  	
	lrCounterGridProd := fbGridCounter.lrTotalCounterEnergy_Production;
	END_IF

END_PROGRAM

// ---- POUs/prgComEffIO.TcPOU
PROGRAM prgComEffIO
VAR
	fbCom		: FB_MqttCommunicator;
END_VAR

fbCom(
	bConnect:= TRUE, 
	sUserName:= '5c5dfa76-f1bb-4218-a3e4-1908f0ce9d03', 
	sUserPassword:= 'aa53ec5d-ecd0-496d-9511-3267225175db', 
	eSavePositionCertificate:= eSavePositionOnPLC.ePostionHardDisk, 
	bConnected=> , 
	bError=> , 
	hrErrorCode=> , 
	eConnectionState=> , 
	eErrorMessage_Out=> );

END_PROGRAM

// ---- POUs/prgRWEffIO.TcPOU
PROGRAM prgRWEffIO
VAR
	fbRW1		: FB_ReadWrite;
END_VAR

fbRW1(bBusy=> , bError=> , udiErrorCodeOut=> , eErrorReadWrite_Out=> );

END_PROGRAM
